PROGRAM MAIN
VAR
	StateMachine: FB_StateMachine;
END_VAR

StateMachine(bUltrasonicSensor:= GVL.bUltrasonicSensor, 
			bUpperLimitSwitch:= GVL.bUpperLimitSwitch, 
			bLowerLimitSwitch:= GVL.bLowerLimitSwitch,
			bPhotocell:= GVL.bPhotocell);
//Scrittura variabili Output
GVL.bMotorUp := StateMachine.bMotorUp;
GVL.bMotorDown := StateMachine.bMotorDown;
GVL.nMotorPosition := GVL.axis.NcToPlc.ActPos;
//Movimentazione motore
GVL.fBPower(Axis:=GVL.axis,
			Enable:=TRUE, 
			Enable_Positive:= GVL.bMotorUp,
			Enable_Negative:= GVL.bMotorDown,
			Override:=100);
GVL.fBJog(Axis:=GVL.axis,
		  JogForward:= GVL.bMotorUp, 
		  JogBackwards:= GVL.bMotorDown, 
		  Velocity:=100);

END_PROGRAM

(* stored: Version 1.1.0.1, ProductVersion 3.1.4024.12
   POU MAIN: Id {cf06fab0-50be-4076-8593-c6c9abf49c38}, SpecialFunc None *)
